(* LS Electric XG5000 project: 23_11_2 *)
(* PLC LSPLC *)

PROGRAM NewProgram (* task: 스캔 프로그램 *)
VAR
    a_t1 : TON;
    t1 : TON;
    t2 : TON;
    t3 : TON;
    t4 : TON;
    t5 : TON;
    t6 : TON;
    t7 : TON;
    t8 : TON;
    램프 : BOOL;
    인풋1 : DWORD := 3811489;
    인풋1_1 : DWORD := 3811488;
    인풋2 : DWORD := 4860066;
    인풋2_1 : DWORD := 4860065;
    인풋3 : DWORD := 8710306;
    인풋3_1 : DWORD;
    인풋4 : DWORD := 8988834;
    인풋4_1 : DWORD := 8726690;
    인풋5 : DWORD := 9048994;
    인풋5_1 : DWORD;
    인풋6 : DWORD := 9053346;
    인풋6_1 : DWORD := 9049250;
    인풋7 : DWORD := 9054286;
    인풋7_1 : DWORD;
    인풋8 : DWORD := 9054354;
    인풋8_1 : DWORD := 9054290;
END_VAR

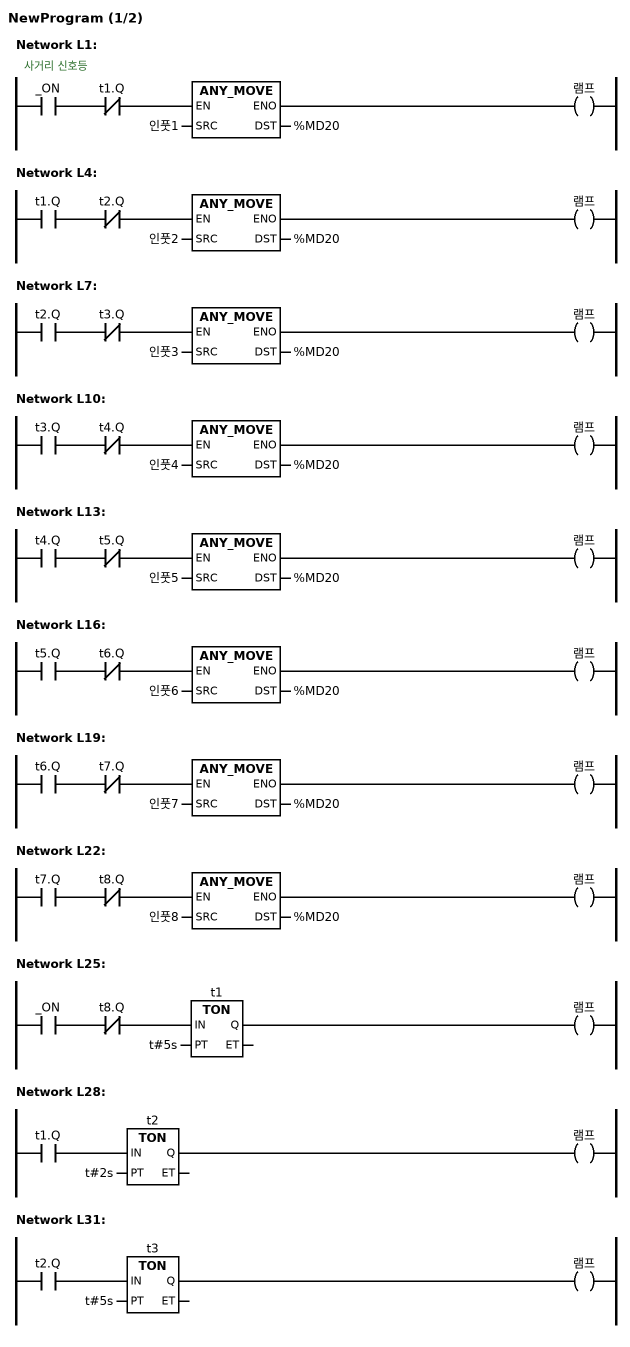
(* 사거리 신호등 *)
(* Rung L1 *)
IF _ON AND NOT t1.Q THEN %MD20 := ANY_MOVE(SRC := 인풋1); END_IF;
램프 := _ON AND NOT t1.Q;
(* Rung L4 *)
IF t1.Q AND NOT t2.Q THEN %MD20 := ANY_MOVE(SRC := 인풋2); END_IF;
램프 := t1.Q AND NOT t2.Q;
(* Rung L7 *)
IF t2.Q AND NOT t3.Q THEN %MD20 := ANY_MOVE(SRC := 인풋3); END_IF;
램프 := t2.Q AND NOT t3.Q;
(* Rung L10 *)
IF t3.Q AND NOT t4.Q THEN %MD20 := ANY_MOVE(SRC := 인풋4); END_IF;
램프 := t3.Q AND NOT t4.Q;
(* Rung L13 *)
IF t4.Q AND NOT t5.Q THEN %MD20 := ANY_MOVE(SRC := 인풋5); END_IF;
램프 := t4.Q AND NOT t5.Q;
(* Rung L16 *)
IF t5.Q AND NOT t6.Q THEN %MD20 := ANY_MOVE(SRC := 인풋6); END_IF;
램프 := t5.Q AND NOT t6.Q;
(* Rung L19 *)
IF t6.Q AND NOT t7.Q THEN %MD20 := ANY_MOVE(SRC := 인풋7); END_IF;
램프 := t6.Q AND NOT t7.Q;
(* Rung L22 *)
IF t7.Q AND NOT t8.Q THEN %MD20 := ANY_MOVE(SRC := 인풋8); END_IF;
램프 := t7.Q AND NOT t8.Q;
(* Rung L25 *)
t1(IN := _ON AND NOT t8.Q, PT := t#5s);
램프 := t1.Q;
(* Rung L28 *)
t2(IN := t1.Q, PT := t#2s);
램프 := t2.Q;
(* Rung L31 *)
t3(IN := t2.Q, PT := t#5s);
램프 := t3.Q;

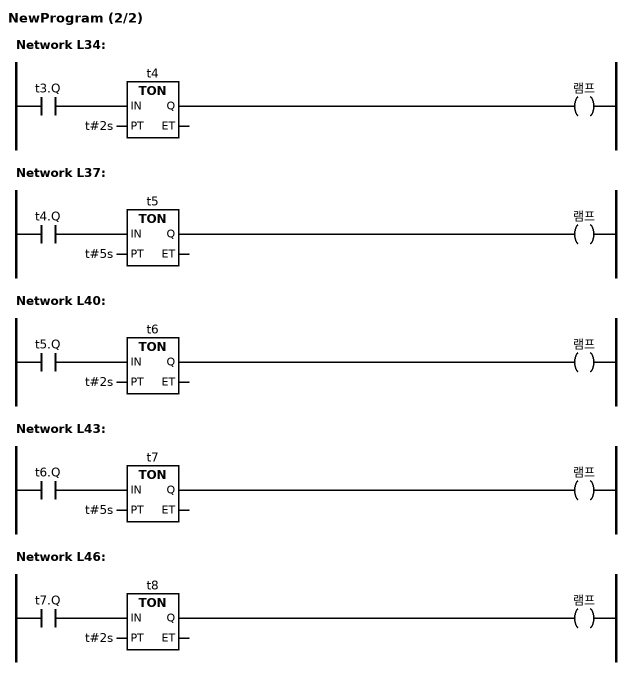
(* Rung L34 *)
t4(IN := t3.Q, PT := t#2s);
램프 := t4.Q;
(* Rung L37 *)
t5(IN := t4.Q, PT := t#5s);
램프 := t5.Q;
(* Rung L40 *)
t6(IN := t5.Q, PT := t#2s);
램프 := t6.Q;
(* Rung L43 *)
t7(IN := t6.Q, PT := t#5s);
램프 := t7.Q;
(* Rung L46 *)
t8(IN := t7.Q, PT := t#2s);
램프 := t8.Q;
END_PROGRAM